Fanuc TP program (LS listing): M_HAND12.LS

/PROG  M_HAND12	  Macro
/ATTR
OWNER		= MNEDITOR;
COMMENT		= "Manual hand12";
PROG_SIZE	= 206;
CREATE		= DATE 28-11-03  TIME 04:31:24;
MODIFIED	= DATE 28-11-03  TIME 04:31:24;
FILE_NAME	= ;
VERSION		= 0;
LINE_COUNT	= 5;
MEMORY_SIZE	= 558;
PROTECT		= READ_WRITE;
TCD:  STACK_SIZE	= 0,
      TASK_PRIORITY	= 50,
      TIME_SLICE	= 0,
      BUSY_LAMP_OFF	= 0,
      ABORT_REQUEST	= 0,
      PAUSE_REQUEST	= 0;
DEFAULT_GROUP	= *,*,*,*,*;
CONTROL_CODE	= 00000000 00000000;
/APPL
/MN
   1:  IF (RO[2:Blowoff ON 1]=ON) THEN ;
   2:  RO[2:Blowoff ON 1]=OFF ;
   3:  ELSE ;
   4:  RO[2:Blowoff ON 1]=ON ;
   5:  ENDIF ;
/POS
/END
